(* Logix 5000 project; controller VET 1756-L62 rev 19.52; software revision 19.01; part 25 of 27 *)
(* tags used below, declared in another part *)
   EColor : DINT[1000];
   Eqp : Equipo[50];
   I : Index;
   RunHours : DINT[1000];
   RunSegs : DINT[1000];
   RunStarts : DINT[1000];
   TabEqp : INT[500];
   _Eqp : Equipo[800];
   _Eqp_Cfg : Eqp_Cfg[800];
   _Origen : Origen[40];
   _Parametros_F : REAL[30];
   _Typlgie : Eqp_Typologie[800];   // Process Flow Typologie
   Batch : batch[10];
   corriente : REAL[40];
   flujometro : flujometro[5];
   peso_tolva : REAL[80];
   Set_Global : DINT[20];
   simulacion : BOOL;
   Timer : TIMER[500];
   Value : DINT[500];
   vdf : VDFS[20];
(* Main1, continued *)

ROUTINE Setup   (* ladder *)
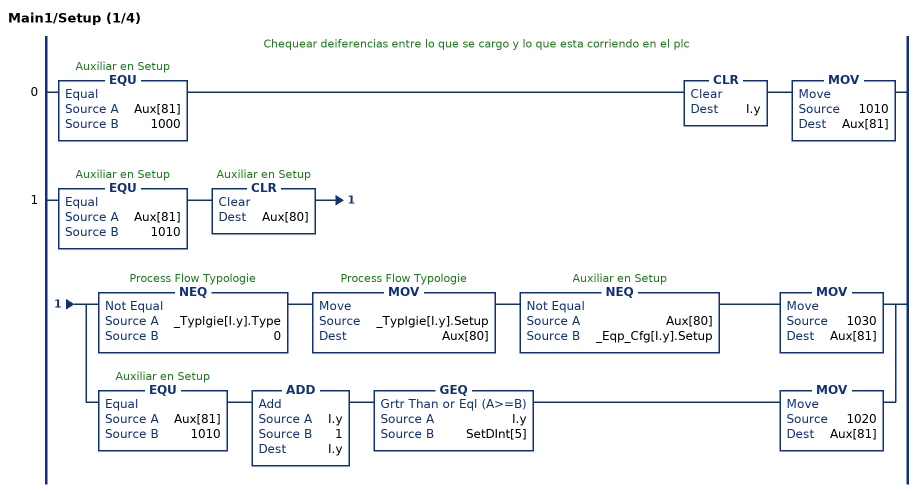
   // Chequear deiferencias entre lo que se cargo y lo que esta corriendo en el plc
   0: EQU(Aux[81],1000)CLR(I.y)MOV(1010,Aux[81]);
   1: EQU(Aux[81],1010)CLR(Aux[80])[NEQ(_Typlgie[I.y].Type,0) MOV(_Typlgie[I.y].Setup,Aux[80]) NEQ(Aux[80],_Eqp_Cfg[I.y].Setup) MOV(1030,Aux[81]) ,EQU(Aux[81],1010) ADD(I.y,1,I.y) GEQ(I.y,SetDInt[5]) MOV(1020,Aux[81]) ];
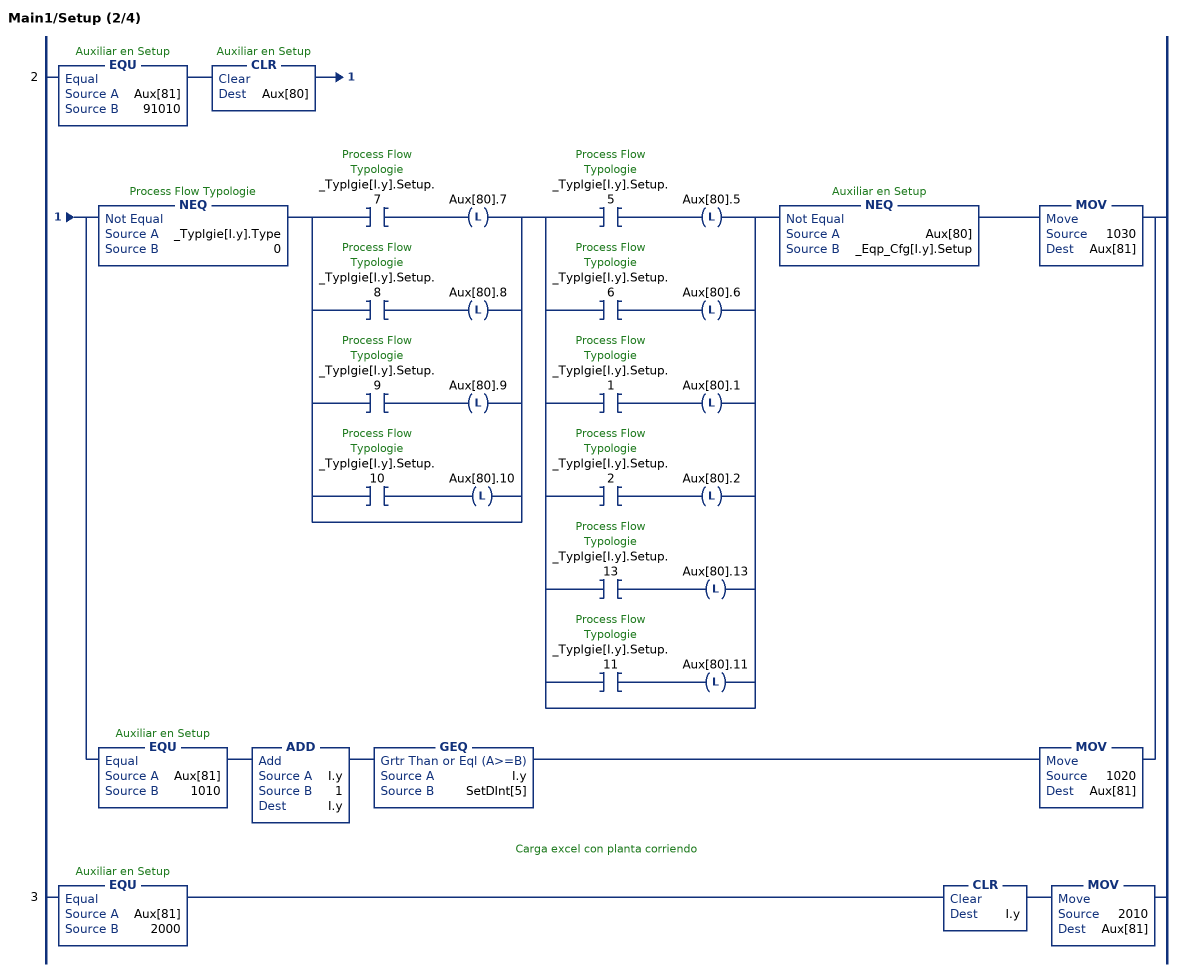
   2: EQU(Aux[81],91010)CLR(Aux[80])[NEQ(_Typlgie[I.y].Type,0) [XIC(_Typlgie[I.y].Setup.7) OTL(Aux[80].7) ,XIC(_Typlgie[I.y].Setup.8) OTL(Aux[80].8) ,XIC(_Typlgie[I.y].Setup.9) OTL(Aux[80].9) ,XIC(_Typlgie[I.y].Setup.10) OTL(Aux[80].10) ,] [XIC(_Typlgie[I.y].Setup.5) OTL(Aux[80].5) ,XIC(_Typlgie[I.y].Setup.6) OTL(Aux[80].6) ,XIC(_Typlgie[I.y].Setup.1) OTL(Aux[80].1) ,XIC(_Typlgie[I.y].Setup.2) OTL(Aux[80].2) ,XIC(_Typlgie[I.y].Setup.13) OTL(Aux[80].13) ,XIC(_Typlgie[I.y].Setup.11) OTL(Aux[80].11) ,] NEQ(Aux[80],_Eqp_Cfg[I.y].Setup) MOV(1030,Aux[81]) ,EQU(Aux[81],1010) ADD(I.y,1,I.y) GEQ(I.y,SetDInt[5]) MOV(1020,Aux[81]) ];
   // Carga excel con planta corriendo
   3: EQU(Aux[81],2000)CLR(I.y)MOV(2010,Aux[81]);
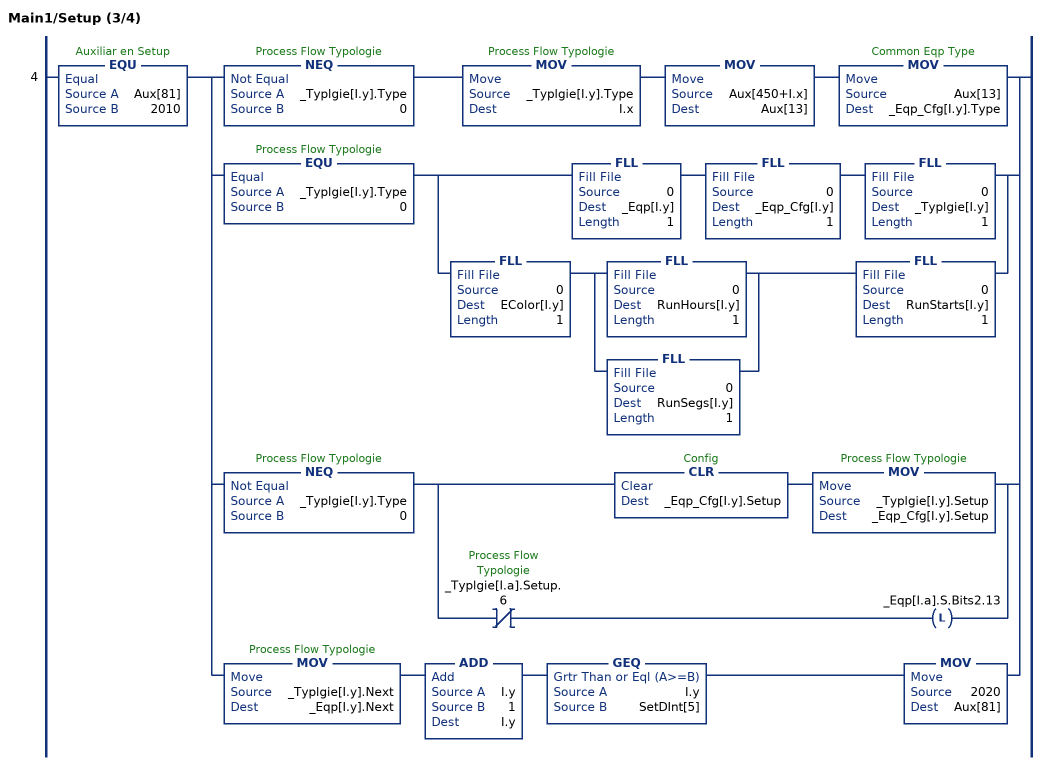
   4: EQU(Aux[81],2010)[NEQ(_Typlgie[I.y].Type,0) MOV(_Typlgie[I.y].Type,I.x) MOV(Aux[450+I.x],Aux[13]) MOV(Aux[13],_Eqp_Cfg[I.y].Type) ,EQU(_Typlgie[I.y].Type,0) [FLL(0,_Eqp[I.y],1) FLL(0,_Eqp_Cfg[I.y],1) FLL(0,_Typlgie[I.y],1) ,FLL(0,EColor[I.y],1) [FLL(0,RunHours[I.y],1) ,FLL(0,RunSegs[I.y],1) ] FLL(0,RunStarts[I.y],1) ] ,NEQ(_Typlgie[I.y].Type,0) [CLR(_Eqp_Cfg[I.y].Setup) MOV(_Typlgie[I.y].Setup,_Eqp_Cfg[I.y].Setup) ,XIO(_Typlgie[I.a].Setup.6) OTL(_Eqp[I.a].S.Bits2.13) ] ,MOV(_Typlgie[I.y].Next,_Eqp[I.y].Next) ADD(I.y,1,I.y) GEQ(I.y,SetDInt[5]) MOV(2020,Aux[81]) ];
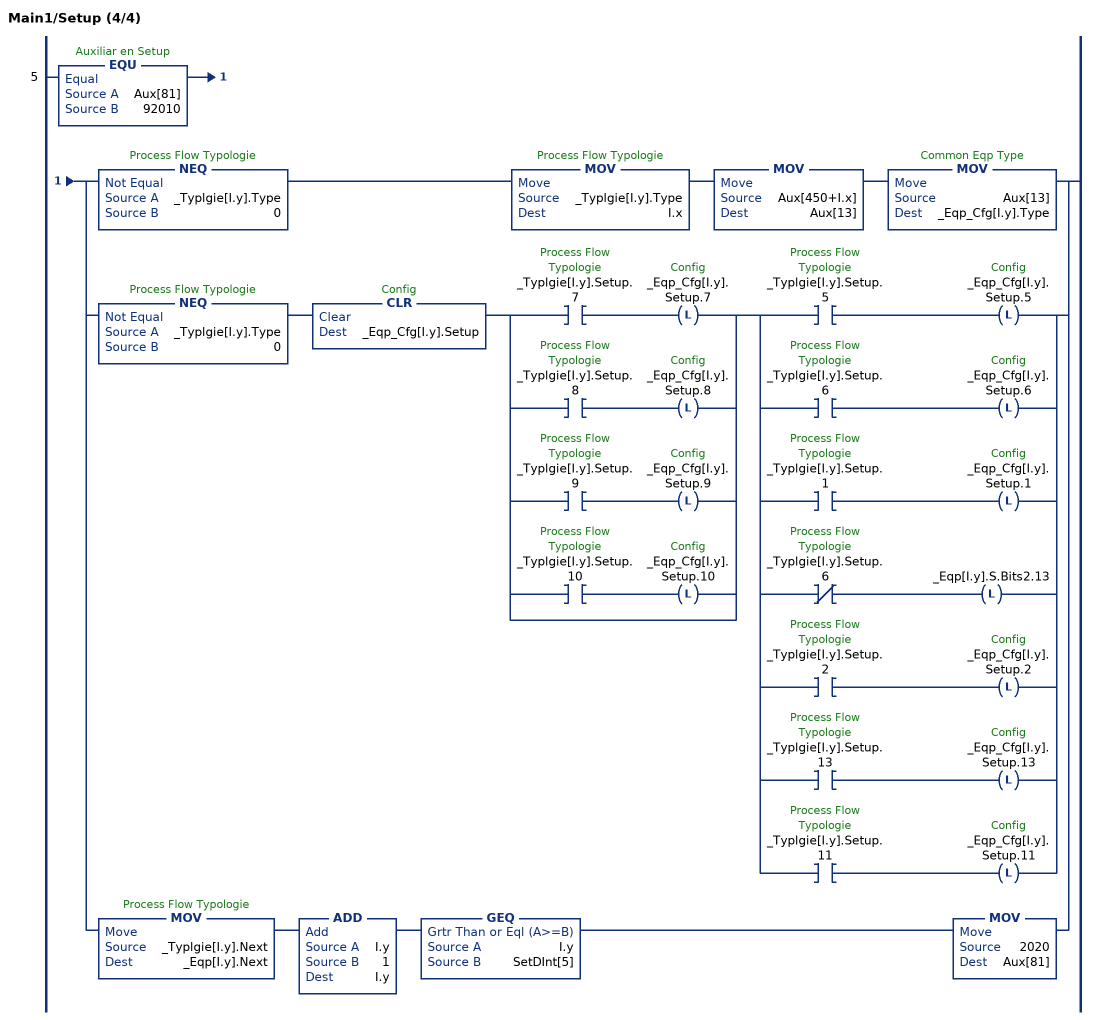
   5: EQU(Aux[81],92010)[NEQ(_Typlgie[I.y].Type,0) MOV(_Typlgie[I.y].Type,I.x) MOV(Aux[450+I.x],Aux[13]) MOV(Aux[13],_Eqp_Cfg[I.y].Type) ,NEQ(_Typlgie[I.y].Type,0) CLR(_Eqp_Cfg[I.y].Setup) [XIC(_Typlgie[I.y].Setup.7) OTL(_Eqp_Cfg[I.y].Setup.7) ,XIC(_Typlgie[I.y].Setup.8) OTL(_Eqp_Cfg[I.y].Setup.8) ,XIC(_Typlgie[I.y].Setup.9) OTL(_Eqp_Cfg[I.y].Setup.9) ,XIC(_Typlgie[I.y].Setup.10) OTL(_Eqp_Cfg[I.y].Setup.10) ,] [XIC(_Typlgie[I.y].Setup.5) OTL(_Eqp_Cfg[I.y].Setup.5) ,XIC(_Typlgie[I.y].Setup.6) OTL(_Eqp_Cfg[I.y].Setup.6) ,XIC(_Typlgie[I.y].Setup.1) OTL(_Eqp_Cfg[I.y].Setup.1) ,XIO(_Typlgie[I.y].Setup.6) OTL(_Eqp[I.y].S.Bits2.13) ,XIC(_Typlgie[I.y].Setup.2) OTL(_Eqp_Cfg[I.y].Setup.2) ,XIC(_Typlgie[I.y].Setup.13) OTL(_Eqp_Cfg[I.y].Setup.13) ,XIC(_Typlgie[I.y].Setup.11) OTL(_Eqp_Cfg[I.y].Setup.11) ] ,MOV(_Typlgie[I.y].Next,_Eqp[I.y].Next) ADD(I.y,1,I.y) GEQ(I.y,SetDInt[5]) MOV(2020,Aux[81]) ];
END_ROUTINE

ROUTINE Startup   (* ladder *)
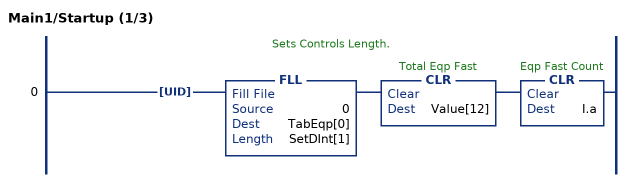
   // Sets Controls Length.
   0: UID()FLL(0,TabEqp[0],SetDInt[1])CLR(Value[12])CLR(I.a);
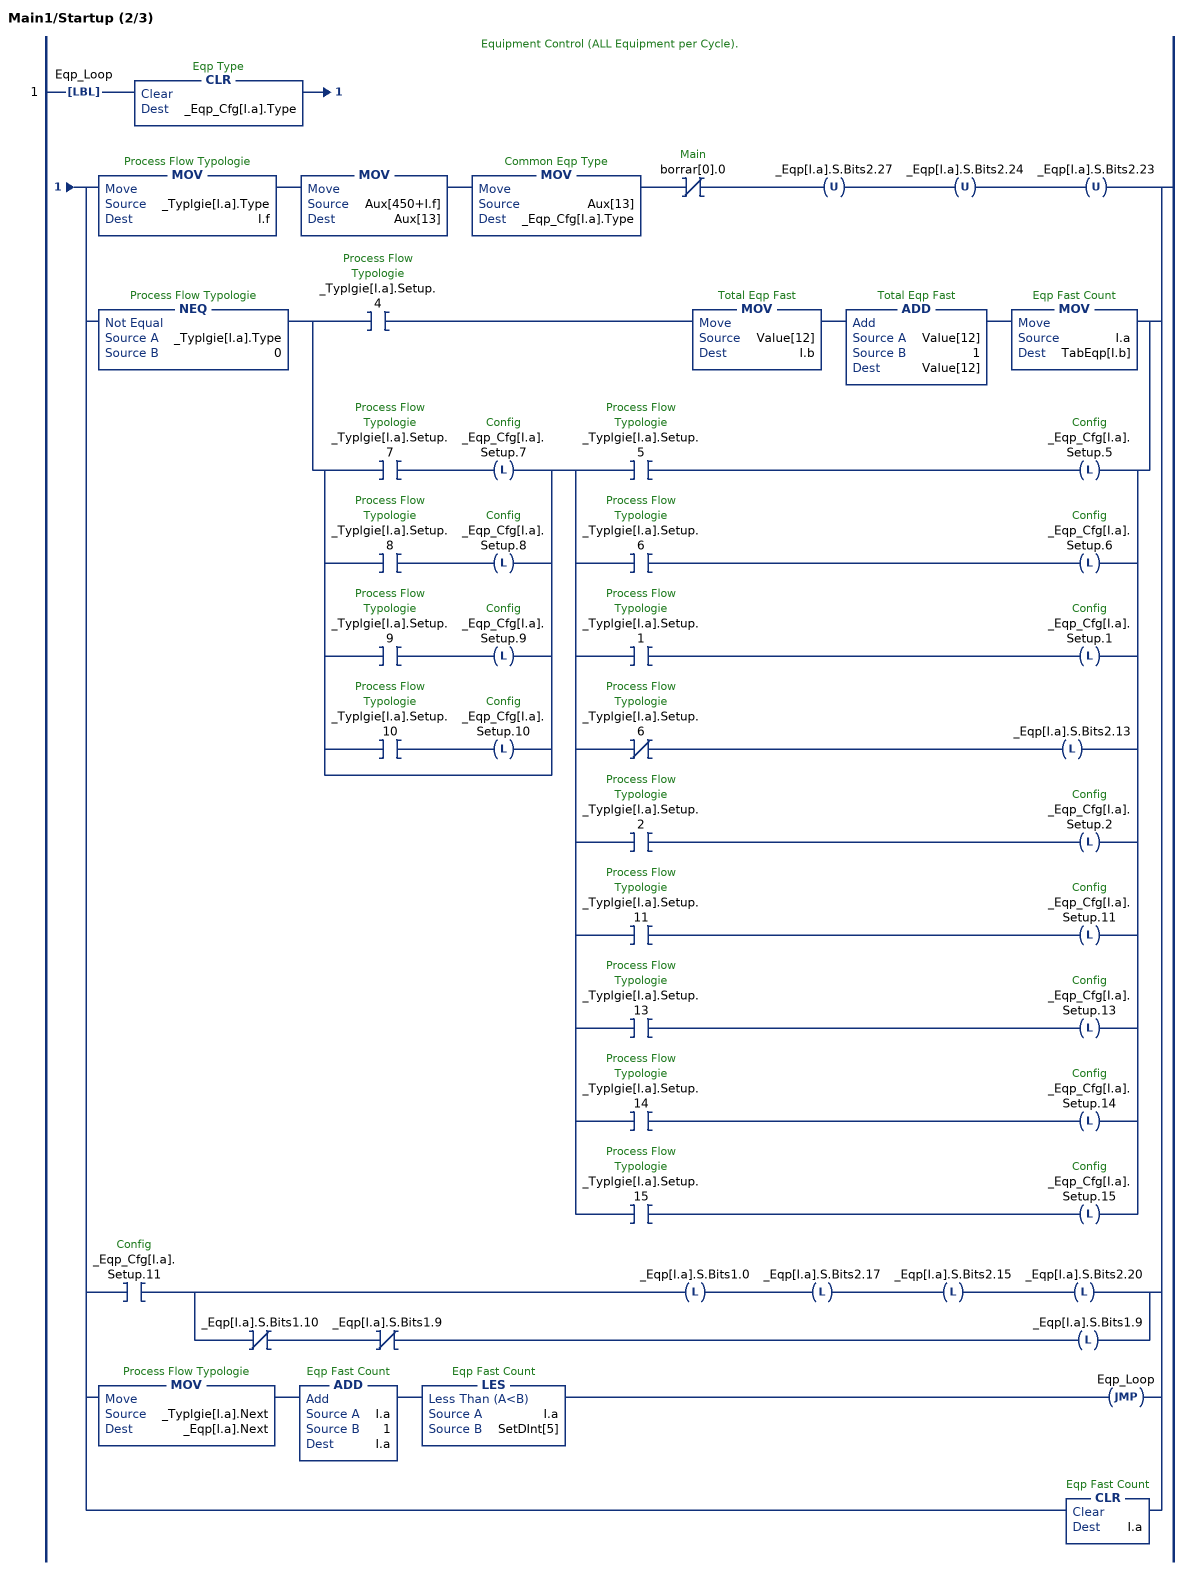
   // Equipment Control (ALL Equipment per Cycle).
   1: LBL(Eqp_Loop)CLR(_Eqp_Cfg[I.a].Type)[MOV(_Typlgie[I.a].Type,I.f) MOV(Aux[450+I.f],Aux[13]) MOV(Aux[13],_Eqp_Cfg[I.a].Type) XIO(borrar[0].0) OTU(_Eqp[I.a].S.Bits2.27) OTU(_Eqp[I.a].S.Bits2.24) OTU(_Eqp[I.a].S.Bits2.23) ,NEQ(_Typlgie[I.a].Type,0) [XIC(_Typlgie[I.a].Setup.4) MOV(Value[12],I.b) ADD(Value[12],1,Value[12]) MOV(I.a,TabEqp[I.b]) ,[XIC(_Typlgie[I.a].Setup.7) OTL(_Eqp_Cfg[I.a].Setup.7) ,XIC(_Typlgie[I.a].Setup.8) OTL(_Eqp_Cfg[I.a].Setup.8) ,XIC(_Typlgie[I.a].Setup.9) OTL(_Eqp_Cfg[I.a].Setup.9) ,XIC(_Typlgie[I.a].Setup.10) OTL(_Eqp_Cfg[I.a].Setup.10) ,] [XIC(_Typlgie[I.a].Setup.5) OTL(_Eqp_Cfg[I.a].Setup.5) ,XIC(_Typlgie[I.a].Setup.6) OTL(_Eqp_Cfg[I.a].Setup.6) ,XIC(_Typlgie[I.a].Setup.1) OTL(_Eqp_Cfg[I.a].Setup.1) ,XIO(_Typlgie[I.a].Setup.6) OTL(_Eqp[I.a].S.Bits2.13) ,XIC(_Typlgie[I.a].Setup.2) OTL(_Eqp_Cfg[I.a].Setup.2) ,XIC(_Typlgie[I.a].Setup.11) OTL(_Eqp_Cfg[I.a].Setup.11) ,XIC(_Typlgie[I.a].Setup.13) OTL(_Eqp_Cfg[I.a].Setup.13) ,XIC(_Typlgie[I.a].Setup.14) OTL(_Eqp_Cfg[I.a].Setup.14) ,XIC(_Typlgie[I.a].Setup.15) OTL(_Eqp_Cfg[I.a].Setup.15) ] ] ,XIC(_Eqp_Cfg[I.a].Setup.11) [OTL(_Eqp[I.a].S.Bits1.0) OTL(_Eqp[I.a].S.Bits2.17) OTL(_Eqp[I.a].S.Bits2.15) OTL(_Eqp[I.a].S.Bits2.20) ,XIO(_Eqp[I.a].S.Bits1.10) XIO(_Eqp[I.a].S.Bits1.9) OTL(_Eqp[I.a].S.Bits1.9) ] ,MOV(_Typlgie[I.a].Next,_Eqp[I.a].Next) ADD(I.a,1,I.a) LES(I.a,SetDInt[5]) JMP(Eqp_Loop) ,CLR(I.a) ];
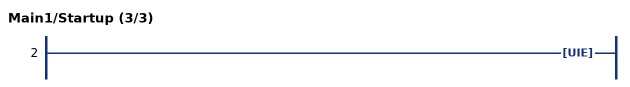
   2: UIE();
END_ROUTINE
END_PROGRAM

PROGRAM Simulacion   (* main routine main *)
VAR
   flujo : REAL[20] := ([0] := 20.0, [1] := 70.0, [2] := 12.0, [3] := 70.0, [4] := 0.4, [5] := 40.0, [6] := 0.4, [7] := 40.0);
        [0]   // Flujo carga Macros
        [1]   // Flujo descarga Macros
        [2]   // Flujo carga Midis
        [3]   // Flujo descarga Midis
        [4]   // Flujo carga Micros 1
        [6]   // Flujo carga Micros 2
        [5]   // Flujo descarga micros 1
        [7]   // Flujo descarga micros 2
   ons : DINT := 1;
   T : TIMER[20] := ([0].PRE := 10000, [0].EN := 1, [0].TT := 1, [1].PRE := 60000, [2].PRE := 60000, [2].ACC := 60000, [2].DN := 1);
END_VAR

ROUTINE main   (* ladder *)
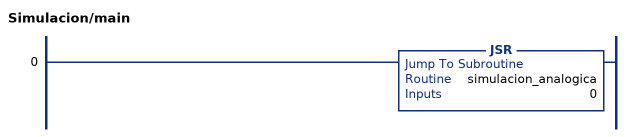
   0: JSR(simulacion_analogica,0);
END_ROUTINE

ROUTINE simulacion_analogica   (* ladder *)
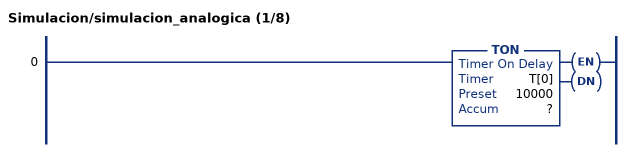
   0: TON(T[0],?,?);
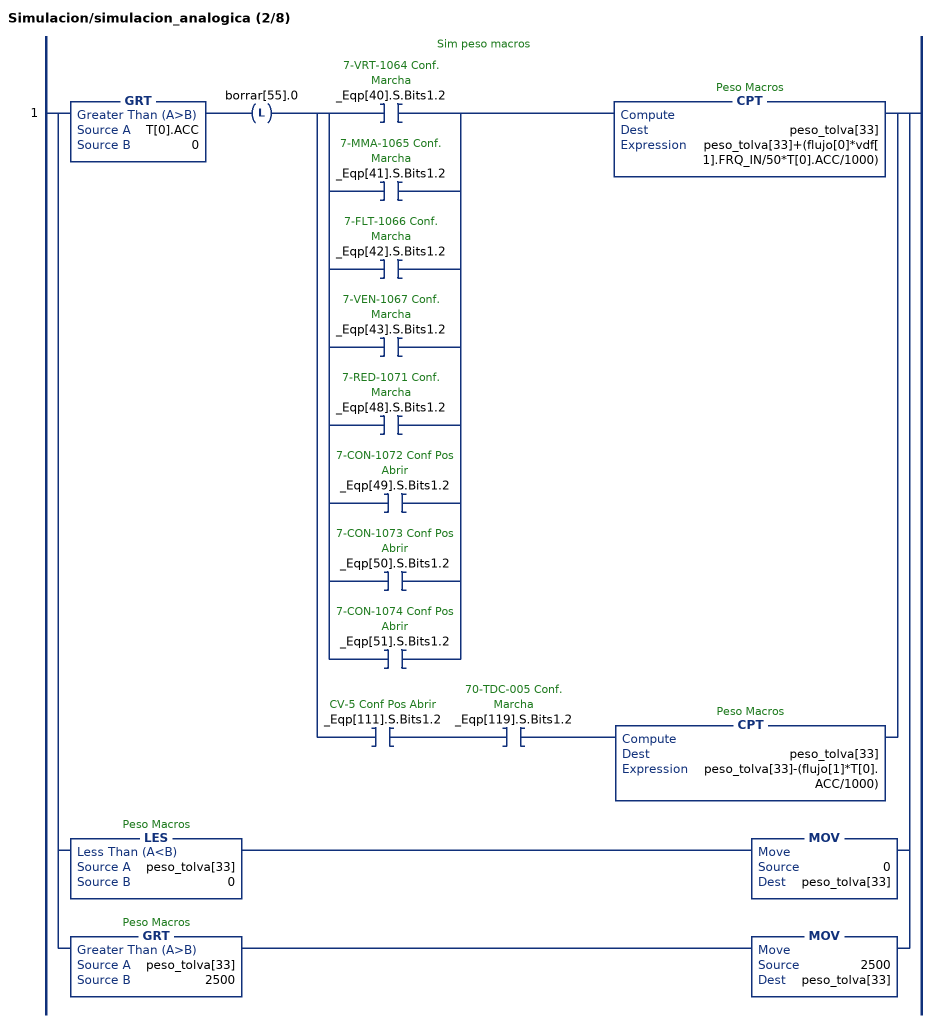
   // Sim peso macros
   1: [GRT(T[0].ACC,0) OTL(borrar[55].0) [[XIC(_Eqp[40].S.Bits1.2) ,XIC(_Eqp[41].S.Bits1.2) ,XIC(_Eqp[42].S.Bits1.2) ,XIC(_Eqp[43].S.Bits1.2) ,XIC(_Eqp[48].S.Bits1.2) ,XIC(_Eqp[49].S.Bits1.2) ,XIC(_Eqp[50].S.Bits1.2) ,XIC(_Eqp[51].S.Bits1.2) ] CPT(peso_tolva[33],peso_tolva[33]+(flujo[0]*vdf[1].FRQ_IN/50*T[0].ACC/1000)) ,XIC(_Eqp[111].S.Bits1.2) XIC(_Eqp[119].S.Bits1.2) CPT(peso_tolva[33],peso_tolva[33]-(flujo[1]*T[0].ACC/1000)) ] ,LES(peso_tolva[33],0) MOV(0,peso_tolva[33]) ,GRT(peso_tolva[33],2500) MOV(2500,peso_tolva[33]) ];
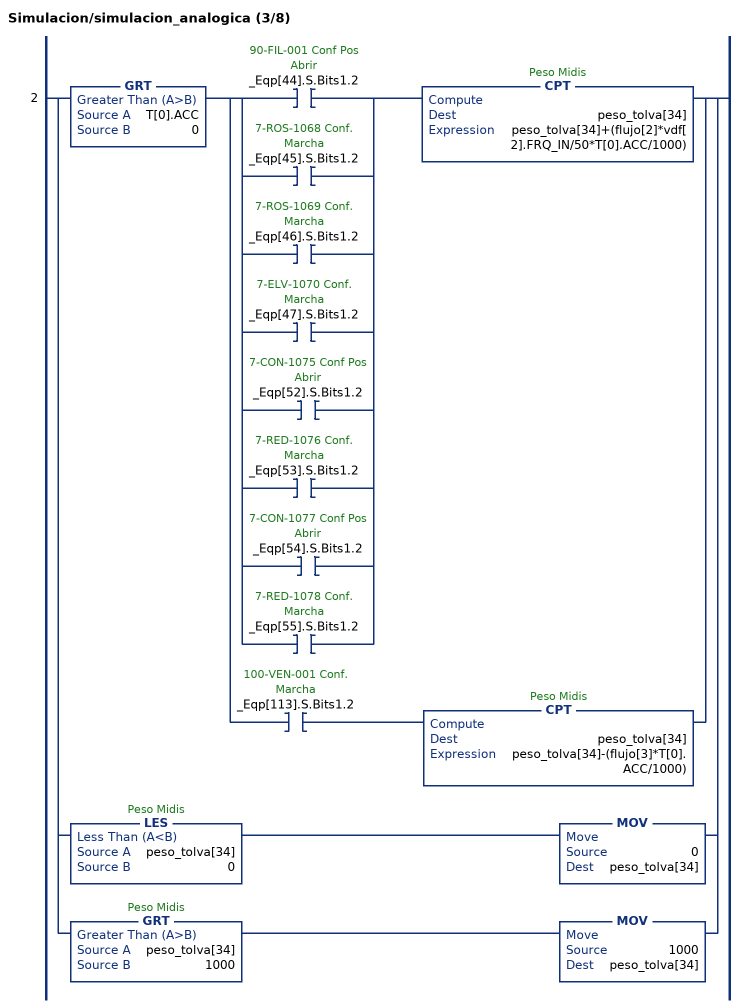
   2: [GRT(T[0].ACC,0) [[XIC(_Eqp[44].S.Bits1.2) ,XIC(_Eqp[45].S.Bits1.2) ,XIC(_Eqp[46].S.Bits1.2) ,XIC(_Eqp[47].S.Bits1.2) ,XIC(_Eqp[52].S.Bits1.2) ,XIC(_Eqp[53].S.Bits1.2) ,XIC(_Eqp[54].S.Bits1.2) ,XIC(_Eqp[55].S.Bits1.2) ] CPT(peso_tolva[34],peso_tolva[34]+(flujo[2]*vdf[2].FRQ_IN/50*T[0].ACC/1000)) ,XIC(_Eqp[113].S.Bits1.2) CPT(peso_tolva[34],peso_tolva[34]-(flujo[3]*T[0].ACC/1000)) ] ,LES(peso_tolva[34],0) MOV(0,peso_tolva[34]) ,GRT(peso_tolva[34],1000) MOV(1000,peso_tolva[34]) ];
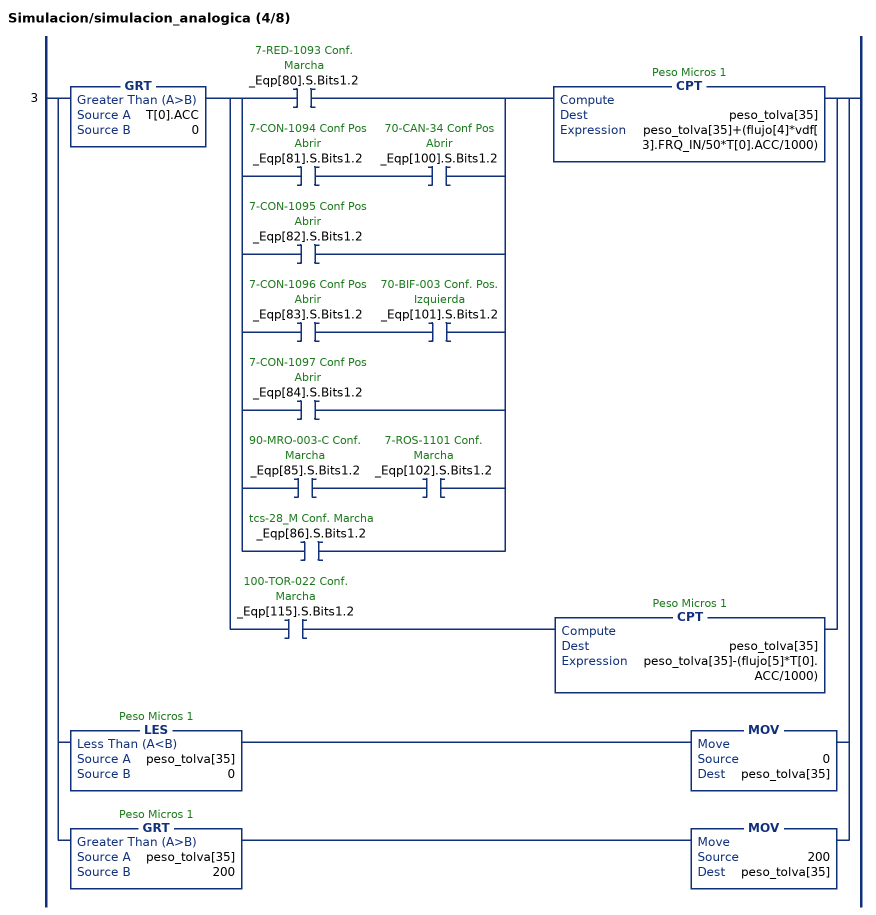
   3: [GRT(T[0].ACC,0) [[XIC(_Eqp[80].S.Bits1.2) ,XIC(_Eqp[81].S.Bits1.2) XIC(_Eqp[100].S.Bits1.2) ,XIC(_Eqp[82].S.Bits1.2) ,XIC(_Eqp[83].S.Bits1.2) XIC(_Eqp[101].S.Bits1.2) ,XIC(_Eqp[84].S.Bits1.2) ,XIC(_Eqp[85].S.Bits1.2) XIC(_Eqp[102].S.Bits1.2) ,XIC(_Eqp[86].S.Bits1.2) ] CPT(peso_tolva[35],peso_tolva[35]+(flujo[4]*vdf[3].FRQ_IN/50*T[0].ACC/1000)) ,XIC(_Eqp[115].S.Bits1.2) CPT(peso_tolva[35],peso_tolva[35]-(flujo[5]*T[0].ACC/1000)) ] ,LES(peso_tolva[35],0) MOV(0,peso_tolva[35]) ,GRT(peso_tolva[35],200) MOV(200,peso_tolva[35]) ];
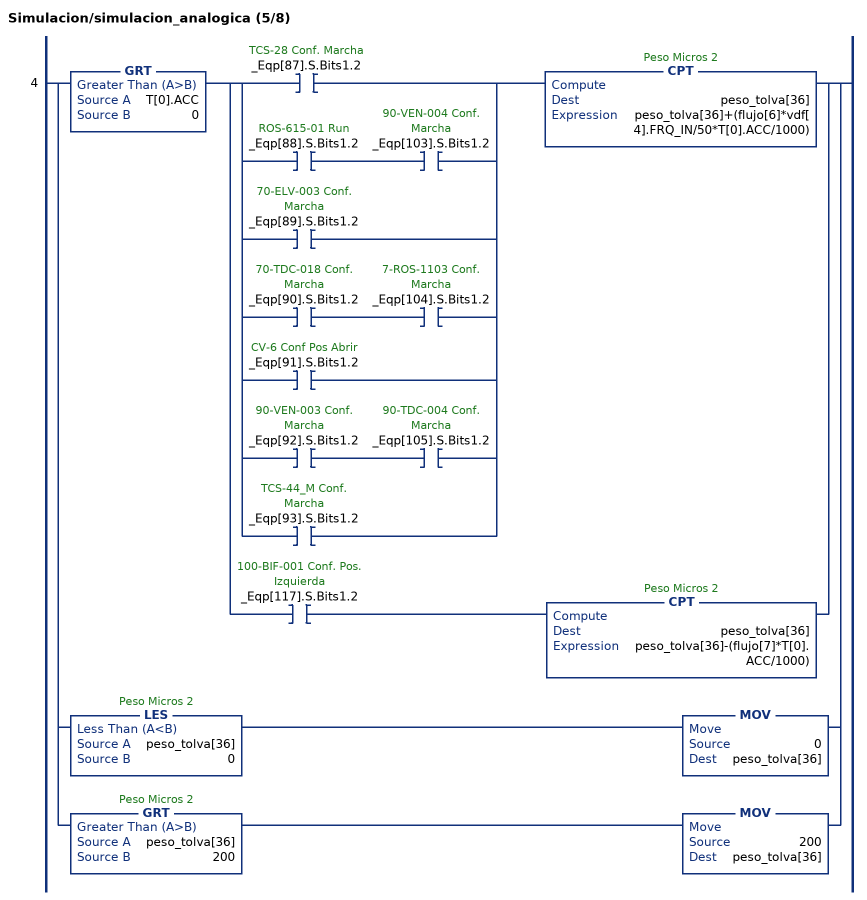
   4: [GRT(T[0].ACC,0) [[XIC(_Eqp[87].S.Bits1.2) ,XIC(_Eqp[88].S.Bits1.2) XIC(_Eqp[103].S.Bits1.2) ,XIC(_Eqp[89].S.Bits1.2) ,XIC(_Eqp[90].S.Bits1.2) XIC(_Eqp[104].S.Bits1.2) ,XIC(_Eqp[91].S.Bits1.2) ,XIC(_Eqp[92].S.Bits1.2) XIC(_Eqp[105].S.Bits1.2) ,XIC(_Eqp[93].S.Bits1.2) ] CPT(peso_tolva[36],peso_tolva[36]+(flujo[6]*vdf[4].FRQ_IN/50*T[0].ACC/1000)) ,XIC(_Eqp[117].S.Bits1.2) CPT(peso_tolva[36],peso_tolva[36]-(flujo[7]*T[0].ACC/1000)) ] ,LES(peso_tolva[36],0) MOV(0,peso_tolva[36]) ,GRT(peso_tolva[36],200) MOV(200,peso_tolva[36]) ];
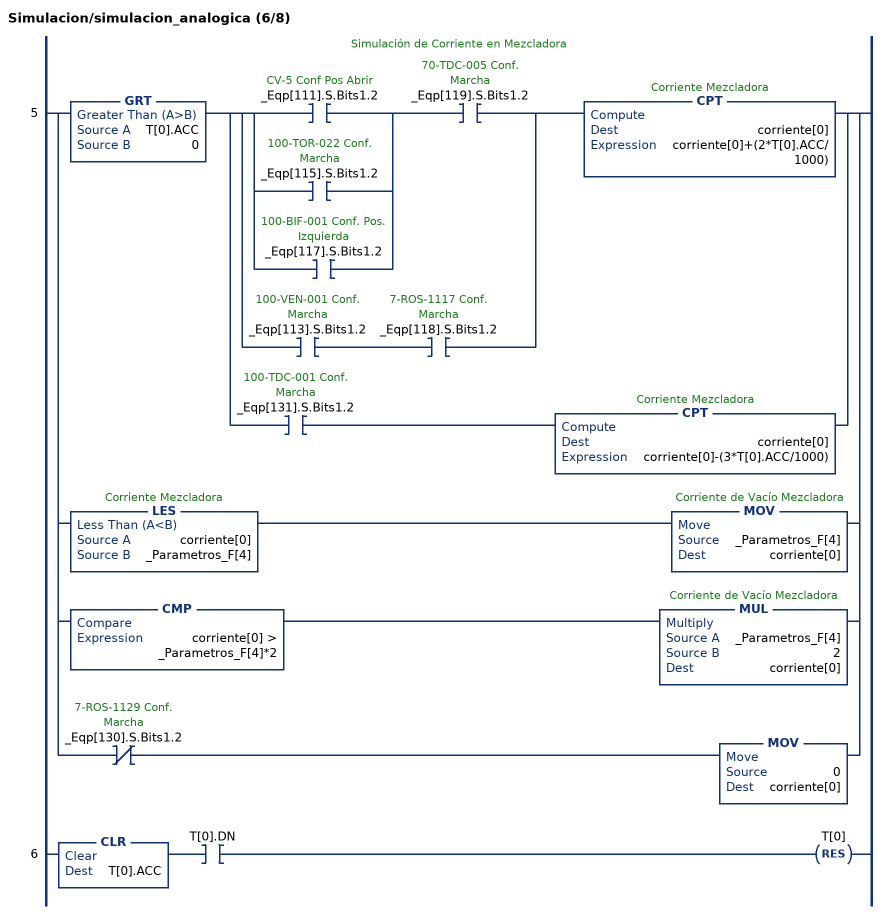
   // Simulación de Corriente en Mezcladora
   5: [GRT(T[0].ACC,0) [[[XIC(_Eqp[111].S.Bits1.2) ,XIC(_Eqp[115].S.Bits1.2) ,XIC(_Eqp[117].S.Bits1.2) ] XIC(_Eqp[119].S.Bits1.2) ,XIC(_Eqp[113].S.Bits1.2) XIC(_Eqp[118].S.Bits1.2) ] CPT(corriente[0],corriente[0]+(2*T[0].ACC/1000)) ,XIC(_Eqp[131].S.Bits1.2) CPT(corriente[0],corriente[0]-(3*T[0].ACC/1000)) ] ,LES(corriente[0],_Parametros_F[4]) MOV(_Parametros_F[4],corriente[0]) ,CMP(corriente[0] > _Parametros_F[4]*2) MUL(_Parametros_F[4],2,corriente[0]) ,XIO(_Eqp[130].S.Bits1.2) MOV(0,corriente[0]) ];
   6: CLR(T[0].ACC)XIC(T[0].DN)RES(T[0]);
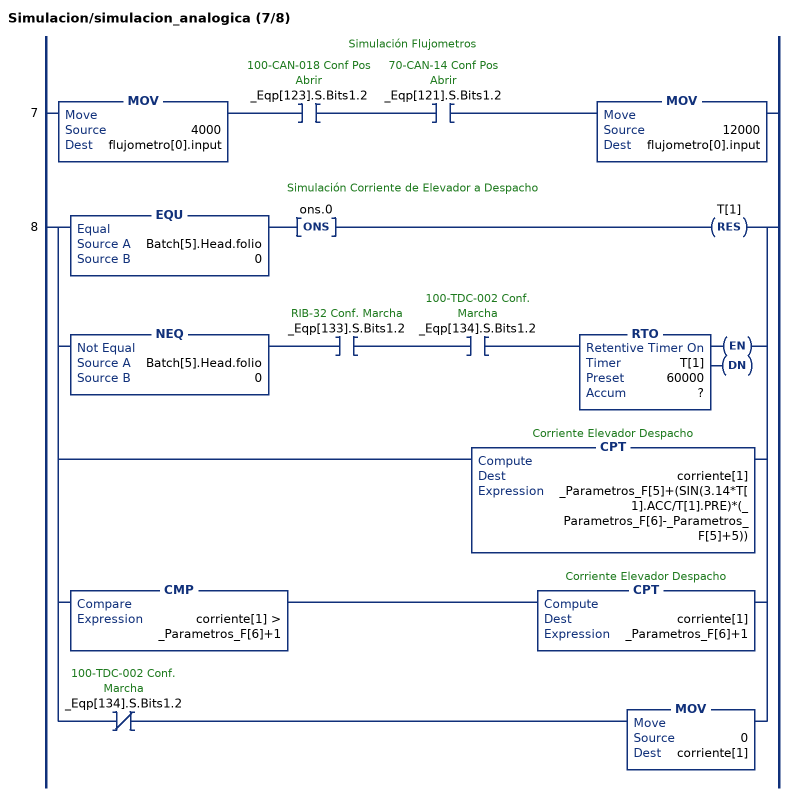
   // Simulación Flujometros
   7: MOV(4000,flujometro[0].input)XIC(_Eqp[123].S.Bits1.2)XIC(_Eqp[121].S.Bits1.2)MOV(12000,flujometro[0].input);
   // Simulación Corriente de Elevador a Despacho
   8: [EQU(Batch[5].Head.folio,0) ONS(ons.0) RES(T[1]) ,NEQ(Batch[5].Head.folio,0) XIC(_Eqp[133].S.Bits1.2) XIC(_Eqp[134].S.Bits1.2) RTO(T[1],?,?) ,CPT(corriente[1],_Parametros_F[5]+(SIN(3.14*T[1].ACC/T[1].PRE)*(_Parametros_F[6]-_Parametros_F[5]+5))) ,CMP(corriente[1] > _Parametros_F[6]+1) CPT(corriente[1],_Parametros_F[6]+1) ,XIO(_Eqp[134].S.Bits1.2) MOV(0,corriente[1]) ];
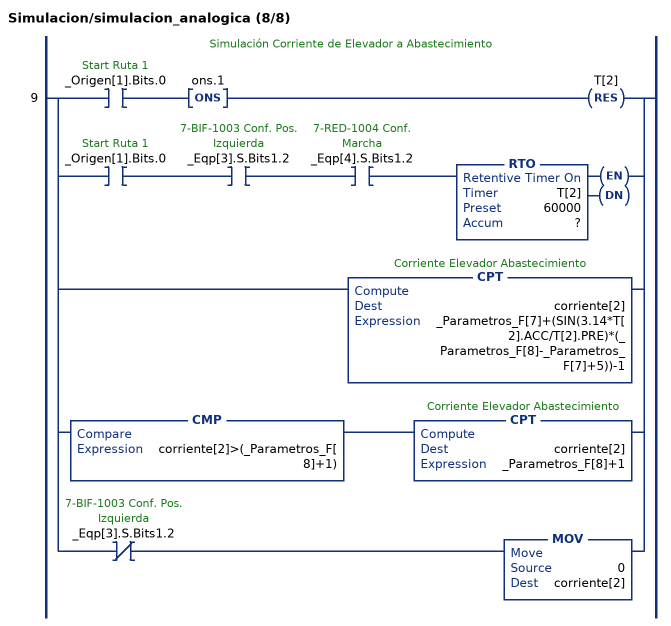
   // Simulación Corriente de Elevador a Abastecimiento
   9: [XIC(_Origen[1].Bits.0) ONS(ons.1) RES(T[2]) ,XIC(_Origen[1].Bits.0) XIC(_Eqp[3].S.Bits1.2) XIC(_Eqp[4].S.Bits1.2) RTO(T[2],?,?) ,CPT(corriente[2],_Parametros_F[7]+(SIN(3.14*T[2].ACC/T[2].PRE)*(_Parametros_F[8]-_Parametros_F[7]+5))-1) ,CMP(corriente[2]>(_Parametros_F[8]+1)) CPT(corriente[2],_Parametros_F[8]+1) ,XIO(_Eqp[3].S.Bits1.2) MOV(0,corriente[2]) ];
END_ROUTINE
END_PROGRAM

PROGRAM Typlgie   (* main routine Main *)
VAR
   _Sel_Comun : Selector := (Idx_eqp := 626, Next[1] := 113, Next[2] := 112, Pos_Real := 1, Pos_Cant := 2, Idx_1Tabeqp := 49);   // Comun selectores
   _Sel_eqp : Sel_eqp[300] := ([1].IDX_SEL := 1, [1].IDX_EQP := 6, [1].POS_CMD[1] := 1, [1].POS_CMD[2] := 1, [1].POS_CMD[3] := 1, [1].POS_CMD[4] := 1, [1].POS_CMD[5] := 1, [1].POS_CMD[6] := 1, [1].POS_CMD[7] := 1, [1].POS_CMD[8] := 1, [1].POS_CMD[9] := 2, [1].POS_CMD[10] := 2, [1].POS_CMD[11] := 2, [1].POS_CMD[12] := 2, [1].POS_CMD[13] := 2, [1].POS_CMD[14] := 2, [1].POS_CMD[15] := 2, [1].POS_CMD[16] := 2, [2].IDX_SEL := 1, [2].IDX_EQP := 7, [2].POS_CMD[1] := 1, [2].POS_CMD[2] := 2, [2].POS_CMD[3] := 3, [2].POS_CMD[4] := 4, [2].POS_CMD[5] := 5, [2].POS_CMD[6] := 6, [2].POS_CMD[7] := 7, [2].POS_CMD[8] := 8, [3].IDX_SEL := 1, [3].IDX_EQP := 8, [3].POS_CMD[9] := 1, [3].POS_CMD[10] := 2, [3].POS_CMD[11] := 3, [3].POS_CMD[12] := 4, [3].POS_CMD[13] := 5, [3].POS_CMD[14] := 6, [3].POS_CMD[15] := 7, [3].POS_CMD[16] := 8, [4].IDX_SEL := 2, [4].IDX_EQP := 138, [4].POS_CMD[1] := 1, [4].POS_CMD[2] := 2);   // Equipos Select
        [14].POS_CMD[4]   // Equipos Select
   _Sel_eqp_comun : Sel_eqp := (IDX_SEL := 6, IDX_EQP := 171, POS_CMD[1] := 1, POS_CMD[2] := 2, POS_CMD[3] := 1);   // Comun equqipos selector
   _Selector : Selector[80] := ([1].Idx_eqp := 170, [1].Next[1] := 20, [1].Next[2] := 21, [1].Next[3] := 22, [1].Next[4] := 23, [1].Next[5] := 24, [1].Next[6] := 25, [1].Next[7] := 26, [1].Next[8] := 27, [1].Next[9] := 28, [1].Next[10] := 29, [1].Next[11] := 30, [1].Next[12] := 31, [1].Next[13] := 32, [1].Next[14] := 33, [1].Next[15] := 34, [1].Next[16] := 35, [1].Pos_Conf := 7, [1].Pos_Cmd := 7, [1].Pos_Real := 7, [1].Pos_Old := 5, [1].Pos_Cant := 16, [1].Idx_1Tabeqp := 1, [1].Timer1.PRE := 10000, [1].Timer2.PRE := 20000, [2].Idx_eqp := 171, [2].Next[1] := 140, [2].Next[2] := 150, [2].Pos_Conf := 2, [2].Pos_Cmd := 2, [2].Pos_Real := 2, [2].Pos_Old := 2, [2].Pos_Cant := 2, [2].Pos_CM := 2, [2].Idx_1Tabeqp := 4, [2].Timer1.PRE := 10000, [2].Timer2.PRE := 20000, [3].Timer1.PRE := 10000, [3].Timer2.PRE := 20000, [4].Timer1.PRE := 10000, [4].Timer2.PRE := 20000, [5].Timer1.PRE := 10000, [5].Timer2.PRE := 20000, [6].Timer1.PRE := 10000, [6].Timer2.PRE := 20000, [7].Timer1.PRE := 10000, [7].Timer2.PRE := 20000, [8].Timer1.PRE := 10000, [8].Timer2.PRE := 20000, [9].Timer1.PRE := 10000, [9].Timer2.PRE := 20000, [10].Timer1.PRE := 10000, [10].Timer2.PRE := 20000, [11].Timer1.PRE := 10000, [11].Timer2.PRE := 20000, [12].Timer1.PRE := 10000, [12].Timer2.PRE := 20000, [13].Timer1.PRE := 10000, [13].Timer2.PRE := 20000, [14].Timer1.PRE := 10000,
        [14].Timer2.PRE := 20000, [15].Timer1.PRE := 10000, [15].Timer2.PRE := 20000, [16].Timer1.PRE := 10000, [16].Timer2.PRE := 20000, [17].Timer1.PRE := 10000, [17].Timer2.PRE := 20000, [18].Timer1.PRE := 10000, [18].Timer2.PRE := 20000, [19].Timer1.PRE := 10000, [19].Timer2.PRE := 20000, [20].Timer1.PRE := 10000, [20].Timer2.PRE := 20000, [21].Timer1.PRE := 10000, [21].Timer2.PRE := 20000, [22].Timer1.PRE := 10000, [22].Timer2.PRE := 20000, [23].Timer1.PRE := 10000, [23].Timer2.PRE := 20000, [24].Timer1.PRE := 10000, [24].Timer2.PRE := 20000, [25].Timer1.PRE := 10000, [25].Timer2.PRE := 20000, [26].Timer1.PRE := 10000, [26].Timer2.PRE := 20000, [27].Timer1.PRE := 10000, [27].Timer2.PRE := 20000, [28].Timer1.PRE := 10000, [28].Timer2.PRE := 20000, [29].Timer1.PRE := 10000, [29].Timer2.PRE := 20000, [30].Timer1.PRE := 10000, [30].Timer2.PRE := 20000, [31].Timer1.PRE := 10000, [31].Timer2.PRE := 20000, [32].Timer1.PRE := 10000, [32].Timer2.PRE := 20000, [33].Timer1.PRE := 10000, [33].Timer2.PRE := 20000, [34].Timer1.PRE := 10000, [34].Timer2.PRE := 20000, [35].Timer1.PRE := 10000, [35].Timer2.PRE := 20000);
   Aux : DINT[40] := ([0] := 35, [1] := 213919, [3] := 190099, [4] := 2427, [5] := 141, [6] := 21, [7] := 21, [8] := 21, [9] := 2, [10] := 26, [11] := 101, [12] := 4, [13] := 1, [14] := 621, [15] := 448, [16] := 328, [18] := 6, [20] := 1, [21] := 2, [22] := 4, [23] := 8, [30] := 1807, [31] := 3104, [32] := 4472, [33] := 9787, [34] := 9442, [35] := 7862, [36] := 1316);
        [0].2   // Suspende verificacion selector
        [6]   // IDX_SEL1_LIM
        [7]   // IDX_SEL2_LIM
        [16]   // Origen Test
        [18]   // Color Equipo Actual
        [0].0   // Pos_deseada_ok
        [0].1   // Pos_read_ok
        [11]   // PTR_EQP7_LIM
        [12]   // Posicion Aux
        [15]   // Destino Final
        [19]   // Color Equipo Next
        [20]   // Posicion Deseada
        [25]   // Posicion Deseada
        [3]   // Count Aux
        [5]   // LIM_PTR1
        [8]   // IDX_SEL_LIM
        [9]   // Pos_cmd_aux
        [10]   // SEL_ACTUAL
        [13]   // IDX_ORIGEN
        [14]   // LIM_PTR5
   Borrar : DINT[100] := ([0] := 2048, [4] := 970, [5] := 993, [6] := 601, [22] := 33735355, [23] := 2, [24] := 2, [34] := 6, [54] := 1, [90] := 40, [97] := 27558, [99] := 617);
   Color_aux : INT[1000] := ([0] := 5, [1] := 5, [2] := 5, [3] := 3, [4] := 2, [5] := 5, [6] := 5, [7] := 5, [8] := 5, [9] := 5, [10] := 2, [11] := 2, [12] := 2, [13] := 2, [14] := 2, [15] := 2, [16] := 5, [17] := 5, [18] := 5, [19] := 5, [20] := 5, [21] := 5, [22] := 5, [23] := 5, [24] := 5, [25] := 5, [26] := 5, [27] := 5, [28] := 5, [29] := 5, [30] := 5, [31] := 5, [32] := 5, [33] := 5, [34] := 5, [35] := 5, [36] := 5, [37] := 5, [38] := 5, [39] := 5, [40] := 3, [41] := 3, [42] := 3, [43] := 3, [44] := 6, [45] := 6, [46] := 6, [47] := 6, [48] := 3, [49] := 3, [50] := 3, [51] := 3, [52] := 6, [53] := 6, [54] := 6, [55] := 6, [56] := 5, [57] := 5, [58] := 5, [59] := 5,
        [60] := 5, [61] := 5, [62] := 5, [63] := 5, [64] := 5, [65] := 5, [66] := 5, [67] := 5, [68] := 5, [69] := 5, [70] := 5, [71] := 5, [72] := 5, [73] := 5, [74] := 5, [75] := 5, [76] := 5, [77] := 5, [78] := 5, [79] := 5, [80] := 4, [81] := 4, [82] := 4, [83] := 4, [84] := 4, [85] := 4, [86] := 4, [87] := 5, [88] := 5, [89] := 5, [90] := 5, [91] := 5, [92] := 5, [93] := 5, [94] := 5, [95] := 5, [96] := 5, [97] := 5, [98] := 5, [99] := 5, [100] := 2, [101] := 2, [102] := 2, [103] := 2, [104] := 2, [105] := 2, [106] := 5, [107] := 5, [108] := 5, [109] := 5, [110] := 5, [111] := 3, [112] := 5, [113] := 6, [114] := 5, [115] := 4, [116] := 5, [117] := 5, [118] := 2, [119] := 2,
        [120] := 5, [121] := 2, [122] := 5, [123] := 5, [124] := 5, [125] := 5, [126] := 6, [127] := 5, [128] := 5, [129] := 5, [131] := 5, [132] := 5, [133] := 6, [134] := 6, [136] := 5, [137] := 6, [138] := 5, [139] := 5, [141] := 5, [142] := 5, [143] := 5, [145] := 5, [147] := 5, [148] := 5, [149] := 5, [151] := 5, [152] := 5, [153] := 5, [154] := 5, [155] := 5, [156] := 5, [157] := 5, [158] := 5, [159] := 5, [160] := 5, [161] := 5, [162] := 5, [163] := 5, [164] := 5, [165] := 5, [166] := 5, [167] := 5, [168] := 5, [169] := 5, [170] := 2, [171] := 6, [172] := 5, [173] := 4, [174] := 4, [175] := 4, [176] := 4, [177] := 4, [178] := 4, [179] := 4, [180] := 4, [181] := 4, [182] := 4, [183] := 4, [184] := 4, [185] := 5,
        [186] := 5, [187] := 4, [188] := 5, [189] := 4, [190] := 2, [191] := 4, [192] := 5, [193] := 4, [194] := 5, [195] := 4, [196] := 5, [197] := 4, [198] := 4, [199] := 5, [200] := 4, [201] := 4, [202] := 5, [203] := 4, [204] := 4, [205] := 5, [206] := 5, [207] := 5, [209] := 4, [210] := 5, [211] := 2, [212] := 4, [213] := 4, [214] := 5, [215] := 2, [216] := 2, [217] := 5, [218] := 2, [219] := 2, [220] := 4, [221] := 2, [222] := 2, [223] := 5, [224] := 4, [225] := 2, [227] := 5, [228] := 2, [229] := 2, [230] := 2, [231] := 4, [232] := 5, [233] := 5, [234] := 5, [235] := 2, [236] := 5, [237] := 2, [238] := 5, [240] := 2, [241] := 5, [244] := 5, [246] := 5, [248] := 2, [249] := 2, [250] := 5, [251] := 2, [252] := 2,
        [253] := 3, [255] := 3, [256] := 3, [257] := 2, [258] := 2, [259] := 5, [262] := 3, [263] := 2, [266] := 5, [268] := 5, [269] := 5, [270] := 5, [271] := 2, [272] := 5, [273] := 5, [274] := 5, [275] := 2, [276] := 5, [277] := 5, [278] := 5, [279] := 2, [280] := 5, [281] := 5, [282] := 5, [283] := 5, [284] := 5, [285] := 5, [287] := 2, [288] := 5, [290] := 2, [291] := 5, [292] := 2, [293] := 2, [294] := 2, [295] := 5, [296] := 5, [297] := 2, [298] := 5, [299] := 2, [300] := 5, [301] := 5, [302] := 2, [303] := 2, [304] := 5, [305] := 2, [306] := 3, [307] := 5, [308] := 2, [309] := 2, [310] := 2, [311] := 2, [312] := 2, [313] := 2, [315] := 2, [316] := 2, [319] := 5, [320] := 5, [321] := 5, [322] := 5, [324] := 2,
        [325] := 2, [326] := 2, [329] := 5, [330] := 5, [331] := 2, [332] := 2, [334] := 2, [335] := 2, [336] := 2, [337] := 5, [338] := 2, [339] := 2, [341] := 5, [342] := 2, [344] := 2, [345] := 5, [346] := 2, [348] := 5, [349] := 2, [350] := 2, [351] := 2, [352] := 2, [353] := 2, [354] := 5, [357] := 2, [358] := 5, [362] := 2, [364] := 5, [367] := 2, [368] := 2, [371] := 5, [372] := 5, [373] := 5, [374] := 2, [376] := 2, [377] := 2, [378] := 2, [379] := 4, [380] := 2, [381] := 2, [383] := 5, [384] := 2, [385] := 5, [386] := 2, [387] := 5, [390] := 5, [391] := 5, [392] := 2, [394] := 2, [395] := 5, [396] := 5, [398] := 2, [399] := 5, [400] := 2, [401] := 5, [402] := 5, [403] := 5, [404] := 5, [405] := 5, [406] := 5,
        [407] := 2, [410] := 5, [411] := 5, [412] := 5, [414] := 2, [415] := 2, [416] := 2, [417] := 5, [418] := 2, [419] := 2, [420] := 5, [422] := 5, [423] := 5, [424] := 5, [425] := 5, [426] := 5, [427] := 2, [429] := 5, [430] := 5, [431] := 5, [432] := 5, [434] := 5, [435] := 5, [436] := 5, [437] := 2, [439] := 5, [440] := 5, [441] := 5, [442] := 5, [443] := 2, [444] := 5, [445] := 5, [446] := 5, [447] := 5, [448] := 5, [450] := 4, [451] := 5, [452] := 5, [453] := 5, [454] := 5, [455] := 5, [456] := 5, [457] := 5, [458] := 5, [459] := 5, [460] := 2, [461] := 5, [462] := 5, [463] := 5, [464] := 5, [465] := 5, [466] := 5, [467] := 2, [468] := 5, [470] := 5, [471] := 5, [472] := 5, [473] := 5, [474] := 2, [475] := 2,
        [476] := 2, [477] := 5, [478] := 2, [479] := 5, [480] := 5, [481] := 5, [482] := 5, [483] := 5, [484] := 5, [485] := 5, [486] := 5, [487] := 5, [488] := 2, [489] := 5, [490] := 5, [491] := 5, [492] := 5, [493] := 5, [494] := 5, [495] := 5, [496] := 5, [497] := 5, [499] := 5, [500] := 5, [501] := 5, [502] := 5, [503] := 5, [504] := 5, [505] := 2, [506] := 5, [507] := 5, [508] := 5, [509] := 5, [510] := 5, [511] := 5, [512] := 5, [513] := 5, [514] := 5, [515] := 5, [516] := 5, [517] := 5, [518] := 5, [520] := 5, [521] := 5, [522] := 5, [525] := 5, [526] := 5, [527] := 5, [528] := 5, [529] := 5, [530] := 5, [531] := 5, [532] := 5, [533] := 5, [534] := 5, [535] := 5, [536] := 5, [537] := 5, [538] := 5, [540] := 5,
        [541] := 5, [542] := 5, [543] := 5, [544] := 2, [545] := 2, [546] := 2, [547] := 5, [548] := 5, [549] := 5, [550] := 1, [551] := 2, [552] := 2, [553] := 5, [554] := 2, [555] := 2, [557] := 5, [558] := 2, [559] := 5, [560] := 3, [561] := 2, [562] := 2, [563] := 5, [564] := 2, [565] := 2, [566] := 2, [567] := 5, [568] := 2, [569] := 5, [571] := 2, [572] := 2, [573] := 2, [574] := 2, [575] := 2, [576] := 2, [577] := 5, [578] := 5, [579] := 5, [580] := 5, [581] := 2, [582] := 5, [583] := 5, [584] := 5, [585] := 5, [586] := 5, [587] := 5, [588] := 5, [589] := 5, [590] := 5, [591] := 2, [592] := 5, [593] := 5, [594] := 5, [595] := 5, [596] := 5, [597] := 5, [598] := 5, [599] := 5, [600] := 5, [601] := 5, [602] := 5,
        [603] := 5, [604] := 2, [607] := 2, [608] := 2, [609] := 2, [611] := 2, [612] := 2, [613] := 2, [614] := 2, [616] := 2, [619] := 2, [620] := 2, [621] := 2, [623] := 2, [627] := 5, [628] := 2, [629] := 2, [630] := 2, [631] := 2, [632] := 7, [633] := 7, [634] := 2, [635] := 2, [636] := 2, [637] := 2, [638] := 2, [640] := 2, [642] := 5, [643] := 5, [644] := 5, [645] := 5, [646] := 5, [647] := 5, [648] := 5, [649] := 5, [650] := 5, [651] := 5, [652] := 5, [653] := 5, [654] := 5, [655] := 5, [656] := 5, [657] := 5, [658] := 5, [659] := 5, [660] := 5, [661] := 5, [662] := 5, [663] := 5, [664] := 5, [665] := 5, [666] := 5, [667] := 5, [668] := 5, [669] := 5, [670] := 5, [671] := 5, [672] := 5, [673] := 5, [674] := 5,
        [675] := 5, [676] := 5, [677] := 5, [678] := 5, [679] := 5, [680] := 5, [681] := 5, [682] := 5, [683] := 5, [684] := 5, [685] := 5, [686] := 5, [687] := 5, [688] := 5, [689] := 5, [690] := 5, [691] := 5, [692] := 5, [693] := 5, [694] := 5, [695] := 5, [696] := 5, [697] := 5, [698] := 5, [699] := 5, [801] := 7, [802] := 7, [803] := 7, [804] := 5, [805] := 5, [806] := 5, [807] := 4, [808] := 4, [809] := 7, [810] := 7, [811] := 7, [812] := 7, [813] := 4, [816] := 5, [820] := 4, [821] := 3, [822] := 2, [823] := 3, [824] := 5, [825] := 2, [826] := 2, [828] := 4, [829] := 3, [830] := 2);
   ecfgcom : Eqp_Cfg := (Type := 8);
        .SETUP.7   // Q1st
        .SETUP.8   // Qseq
   eqpcom : Equipo := (S.Bits1 := 1041, S.Bits2 := 136810501);   // Comun Equipos
        .S.BITS1.10   // ILH
        .S.BITS2.2   // Bit SUSP_VERIF
        .TIMER.TPO1.DN   // CMRET
        .TIMER.TPO2.DN   // OMRRET
        .S.BITS2.9   // LH_SUS
        .S.BITS2.13   // ENC_SIG
        .S.BITS2.24   // OMR
        .S.BITS3.0   // BWD RX 1
        .S.BITS3.1   // BWD RX 2
        .S.BITS3.2   // BWD RX 3
        .S.BITS3.3   // BWD RX 4
        .S.BITS3.4   // BWD TX 1
        .S.BITS3.5   // BWD TX 2
        .S.BITS3.8   // FWD RX 1
        .S.BITS3.9   // FWD RX 2
        .S.BITS3.10   // FWD RX 3
        .S.BITS3.11   // FWD RX 4
        .S.BITS3.12   // FWD TX 1
        .S.BITS3.13   // FWD TX 2
        .S.BITS3.14   // FWD TX 3
        .S.BITS3.15   // FWD TX 4
        .S.BITS3.16   // PROCESADO
        .S.BITS3.18   // Q1st aux
        .S.BITS3.19   // Qseq aux
        .S.BITS2.3   // CM AUX SELECTOR
        .S.BITS1.2   // CM
   OrigCom2 : Origen := (_1eqp := 133, Bits := 1, Color := 6, DestReal := 150, DestOld := 150, DestNew := 2, Tespera.PRE := 120000);
        .BITS.0   // OMR ON
        .BITS.1   // OMR OFF
        .DESTFIN   // Destino Final Real
        .BITS.4   // Test Ruta Actual
        .BITS.6   // Product Mismatch
        .BITS.5   // Destino Real
        .BITS.2   // Cambiar a Ruta New
        .PROD1EQP   // Codigo Prod Inic
        .PRODFIN   // Codigo Prod Final
        .DESTREAL   // Destino Final Real
        .PROD1EQPIND   // Index Prod Inic
        .PRODFININD   // Index Prod Final
        .BITS.3   // Processing Ruta
        .BITS.7   // Enclavamiento Externo Cambios
        .BITS.8   // Comando Primario de Cambio
   SetDInt : DINT[500] := ([1] := 620, [4] := 20, [5] := 18, [6] := 100, [7] := 11, [9] := 5);
   Table1 : DINT[100] := ([0] := 1, [1] := 2, [2] := 4, [3] := 8);
   ti : Index := (a := 3, b := 4, c := 3, d := 3, e := 3, f := 300, g := 171, h := 5, i := 35, j := 300, k := 300, l := 35, m := 2, n := 2, o := 2, p := 150, r := 171, s := 133, t := 2, u := 150, z := 2, a1 := 134, b1 := 2, c1 := 2, d1 := 138, e1 := 2, f1 := 171, m1 := 2, a2 := 150);
        .D   // IDX_SEL1
        .F   // PTR_EQP1
        .H   // PTR_EQP_SEL
        .I   // PTR_EQP2
        .J   // PTR_EQP6
        .K   // PTR_EQP7
        .L   // PTR_EQP_SIG
        .M   // Posicion Real
        .Y   // Indice Batch
        .Z   // Indice Origen
        .A1   // Idx_Eqp
        .B1   // Sel Pos Fut
        .F1   // Indx Selector en Eqp
        .B   // Fase procesamiento secuencias
        .E   // Loop Selector Indx
        .N   // Posicion Comando
        .O   // Pos. Nueva o Test
        .Q   // Code Prod Inic Indx
        .T   // Indice Destino
        .U   // Destino Deseado
        .A   // Fases Ejecucion Topologia
        .V   // Indice Selector
        .W   // Indice Eqp Dest
        .X   // Code Prod Fin Indx
        .E1   // Pos. Real Selector
        .A2   // Eqp Sgte Futuro
        .C   // IDX_SEL
        .G   // PTR_EQP
END_VAR

ROUTINE Eqp_Propag   (* ladder *)
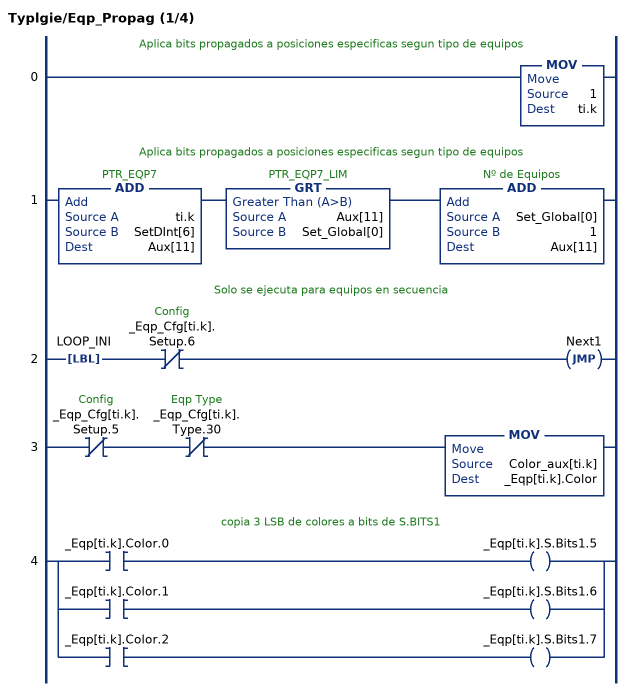
   // Aplica bits propagados a posiciones especificas segun tipo de equipos
   0: MOV(1,ti.k);
   // Aplica bits propagados a posiciones especificas segun tipo de equipos
   1: ADD(ti.k,SetDInt[6],Aux[11])GRT(Aux[11],Set_Global[0])ADD(Set_Global[0],1,Aux[11]);
   // Solo se ejecuta para equipos en secuencia
   2: LBL(LOOP_INI)XIO(_Eqp_Cfg[ti.k].Setup.6)JMP(Next1);
   3: XIO(_Eqp_Cfg[ti.k].Setup.5)XIO(_Eqp_Cfg[ti.k].Type.30)MOV(Color_aux[ti.k],_Eqp[ti.k].Color);
   // copia 3 LSB de colores a bits de S.BITS1
   4: [XIC(_Eqp[ti.k].Color.0) OTE(_Eqp[ti.k].S.Bits1.5) ,XIC(_Eqp[ti.k].Color.1) OTE(_Eqp[ti.k].S.Bits1.6) ,XIC(_Eqp[ti.k].Color.2) OTE(_Eqp[ti.k].S.Bits1.7) ];
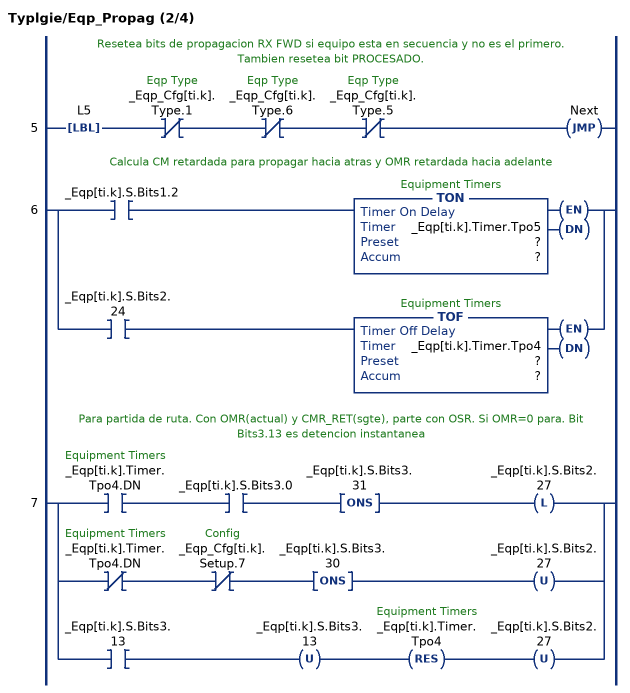
   // Resetea bits de propagacion RX FWD si equipo esta en secuencia y no es el primero. Tambien resetea bit PROCESADO.
   5: LBL(L5)XIO(_Eqp_Cfg[ti.k].Type.1)XIO(_Eqp_Cfg[ti.k].Type.6)XIO(_Eqp_Cfg[ti.k].Type.5)JMP(Next);
   // Calcula CM retardada para propagar hacia atras y OMR retardada hacia adelante
   6: [XIC(_Eqp[ti.k].S.Bits1.2) TON(_Eqp[ti.k].Timer.Tpo5,?,?) ,XIC(_Eqp[ti.k].S.Bits2.24) TOF(_Eqp[ti.k].Timer.Tpo4,?,?) ];
   // Para partida de ruta. Con OMR(actual) y CMR_RET(sgte), parte con OSR. Si OMR=0 para. Bit Bits3.13 es detencion instantanea
   7: [XIC(_Eqp[ti.k].Timer.Tpo4.DN) XIC(_Eqp[ti.k].S.Bits3.0) ONS(_Eqp[ti.k].S.Bits3.31) OTL(_Eqp[ti.k].S.Bits2.27) ,XIO(_Eqp[ti.k].Timer.Tpo4.DN) XIO(_Eqp_Cfg[ti.k].Setup.7) ONS(_Eqp[ti.k].S.Bits3.30) OTU(_Eqp[ti.k].S.Bits2.27) ,XIC(_Eqp[ti.k].S.Bits3.13) OTU(_Eqp[ti.k].S.Bits3.13) RES(_Eqp[ti.k].Timer.Tpo4) OTU(_Eqp[ti.k].S.Bits2.27) ];
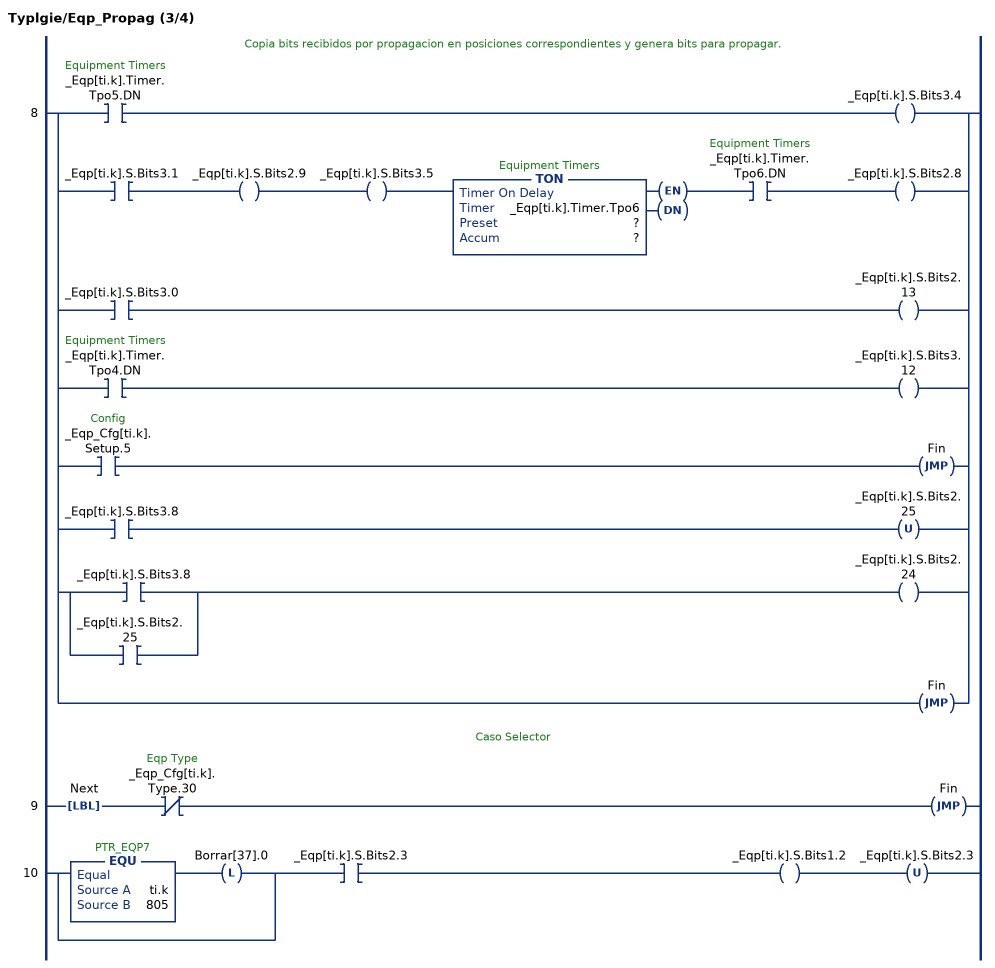
   // Copia bits recibidos por propagacion en posiciones correspondientes y genera bits para propagar.
   8: [XIC(_Eqp[ti.k].Timer.Tpo5.DN) OTE(_Eqp[ti.k].S.Bits3.4) ,XIC(_Eqp[ti.k].S.Bits3.1) OTE(_Eqp[ti.k].S.Bits2.9) OTE(_Eqp[ti.k].S.Bits3.5) TON(_Eqp[ti.k].Timer.Tpo6,?,?) XIC(_Eqp[ti.k].Timer.Tpo6.DN) OTE(_Eqp[ti.k].S.Bits2.8) ,XIC(_Eqp[ti.k].S.Bits3.0) OTE(_Eqp[ti.k].S.Bits2.13) ,XIC(_Eqp[ti.k].Timer.Tpo4.DN) OTE(_Eqp[ti.k].S.Bits3.12) ,XIC(_Eqp_Cfg[ti.k].Setup.5) JMP(Fin) ,XIC(_Eqp[ti.k].S.Bits3.8) OTU(_Eqp[ti.k].S.Bits2.25) ,[XIC(_Eqp[ti.k].S.Bits3.8) ,XIC(_Eqp[ti.k].S.Bits2.25) ] OTE(_Eqp[ti.k].S.Bits2.24) ,JMP(Fin) ];
   // Caso Selector
   9: LBL(Next)XIO(_Eqp_Cfg[ti.k].Type.30)JMP(Fin);
   10: [EQU(ti.k,805) OTL(Borrar[37].0) ,]XIC(_Eqp[ti.k].S.Bits2.3)OTE(_Eqp[ti.k].S.Bits1.2)OTU(_Eqp[ti.k].S.Bits2.3);
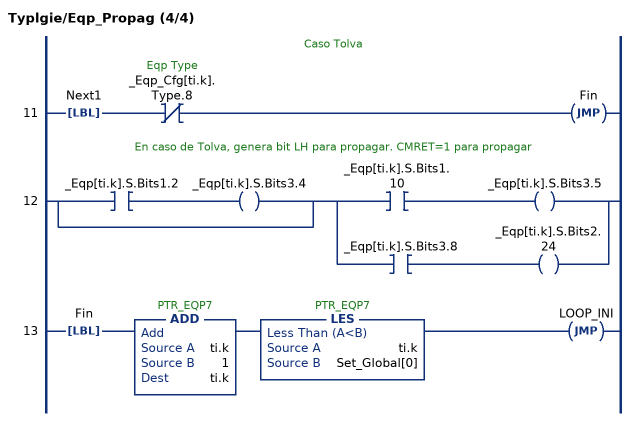
   // Caso Tolva
   11: LBL(Next1)XIO(_Eqp_Cfg[ti.k].Type.8)JMP(Fin);
   // En caso de Tolva, genera bit LH para propagar. CMRET=1 para propagar
   12: [XIC(_Eqp[ti.k].S.Bits1.2) OTE(_Eqp[ti.k].S.Bits3.4) ,][XIC(_Eqp[ti.k].S.Bits1.10) OTE(_Eqp[ti.k].S.Bits3.5) ,XIC(_Eqp[ti.k].S.Bits3.8) OTE(_Eqp[ti.k].S.Bits2.24) ];
   13: LBL(Fin)ADD(ti.k,1,ti.k)LES(ti.k,Set_Global[0])JMP(LOOP_INI);
END_ROUTINE
